_CFC_ (* Continuous Function Chart, elements in execution order *)
#0 OR(SHU6_PV1_YA4_UP_RESET, SHU6_PV1_SB)
#1 SEL(SHU6_PV1_YA4_AI1_FILTER_ON, T#0ms, T#2s)
#2 fb_YA3:ISTOK_ANALOGVH(enable: TRUE, rawValue: SHU6_PV1_1YA4_AI5, reset: #0, enableLimitCtrl: TRUE, ctrlVoltage: NOT SHU6_PV1_YA4_AI1_CVOLT, changeValueWithoutPower: TRUE, highRange: YA_HIGHRANGE, lowRange: YA_LOWRANGE, highLimit: SHU6_PV1_YA_HIGHLIMIT, lowLimit: SHU6_PV1_YA_LOWLIMIT, filterTime: #1, offset: ofset, delayEnable: YA_DELAY)
#3 SHU6_PV1_YA4_UP_VN <= #2.presentValue
#4 SHU6_PV1_YA4_UP_DOST <= #2.reliability
#5 Lt_otkr_zakr:ISTOK_LT(dost: #2.reliability, x: #2.presentValue, ust: 5, shkal: -, gist: 3)
#6 SHU6_PV1_YA4_ZKR <= #5.Xm
#7 gt_otkr_otr:ISTOK_GT(dost: #2.reliability, x: #2.presentValue, ust: 95, shkal: -, gist: 3)
#8 SHU6_PV1_YA4_OTK <= #7.Xb
#9 SUB(YA4_UST_VKL_STER_REG, YA4_UST_OTKL_STER_REG)
#10 fb_YA3bUST_VKL_STER_REG:ISTOK_GT(dost: #2.reliability, x: #2.presentValue, ust: YA4_UST_VKL_STER_REG, shkal: -, gist: #9)
#11 SHU6_PV1_YA4_B_UST_VKL_STER_REG <= #10.Xb
#12 SHU6_PV1_YA4_M_UST_VKL_STER_REG <= #10.XbN
#13 SUB(YA4_UST_OTKL_UVEL_CHAST, YA4_UST_VKL_UVEL_CHAST)
#14 fb_YA3mOTKL_STER_REG:ISTOK_LT(dost: #2.reliability, x: #2.presentValue, ust: YA4_UST_VKL_UVEL_CHAST, shkal: -, gist: #13)
#15 SHU6_PV1_YA4_M_UST_VKL_UVEL_CHAST <= #14.Xm
#16 SHU6_PV1_YA4_B_UST_VKL_UVEL_CHAST <= #14.XmN
_END_CFC_
(* the same logic as Structured Text *)
fb_YA3(enable := TRUE, rawValue := SHU6_PV1_1YA4_AI5, reset := SHU6_PV1_YA4_UP_RESET OR SHU6_PV1_SB, enableLimitCtrl := TRUE, ctrlVoltage := NOT SHU6_PV1_YA4_AI1_CVOLT, changeValueWithoutPower := TRUE, highRange := YA_HIGHRANGE, lowRange := YA_LOWRANGE, highLimit := SHU6_PV1_YA_HIGHLIMIT, lowLimit := SHU6_PV1_YA_LOWLIMIT, filterTime := SEL(SHU6_PV1_YA4_AI1_FILTER_ON, T#0ms, T#2s), offset := ofset, delayEnable := YA_DELAY);
SHU6_PV1_YA4_UP_VN := fb_YA3.presentValue;
SHU6_PV1_YA4_UP_DOST := fb_YA3.reliability;
Lt_otkr_zakr(dost := fb_YA3.reliability, x := fb_YA3.presentValue, ust := 5, gist := 3);
SHU6_PV1_YA4_ZKR := Lt_otkr_zakr.Xm;
gt_otkr_otr(dost := fb_YA3.reliability, x := fb_YA3.presentValue, ust := 95, gist := 3);
SHU6_PV1_YA4_OTK := gt_otkr_otr.Xb;
fb_YA3bUST_VKL_STER_REG(dost := fb_YA3.reliability, x := fb_YA3.presentValue, ust := YA4_UST_VKL_STER_REG, gist := YA4_UST_VKL_STER_REG - YA4_UST_OTKL_STER_REG);
SHU6_PV1_YA4_B_UST_VKL_STER_REG := fb_YA3bUST_VKL_STER_REG.Xb;
SHU6_PV1_YA4_M_UST_VKL_STER_REG := fb_YA3bUST_VKL_STER_REG.XbN;
fb_YA3mOTKL_STER_REG(dost := fb_YA3.reliability, x := fb_YA3.presentValue, ust := YA4_UST_VKL_UVEL_CHAST, gist := YA4_UST_OTKL_UVEL_CHAST - YA4_UST_VKL_UVEL_CHAST);
SHU6_PV1_YA4_M_UST_VKL_UVEL_CHAST := fb_YA3mOTKL_STER_REG.Xm;
SHU6_PV1_YA4_B_UST_VKL_UVEL_CHAST := fb_YA3mOTKL_STER_REG.XmN;
END_PROGRAM

(* POU Input/CI/MP1_OB, CFC *)
PROGRAM MP1_OB
VAR
	fb_M1_OBRbSM: ISTOK_GT;
	fb_M1b30: ISTOK_GT;
	fb_M1_OBRb45: ISTOK_GT;
	fb_M1_OBRm0_1: ISTOK_LT;
	fb_M_OBR: ISTOK_ANALOGVH;
	ofset: INT := 0;
	SR_DOST_M1: RS;
	dost_ton: TON;
END_VAR
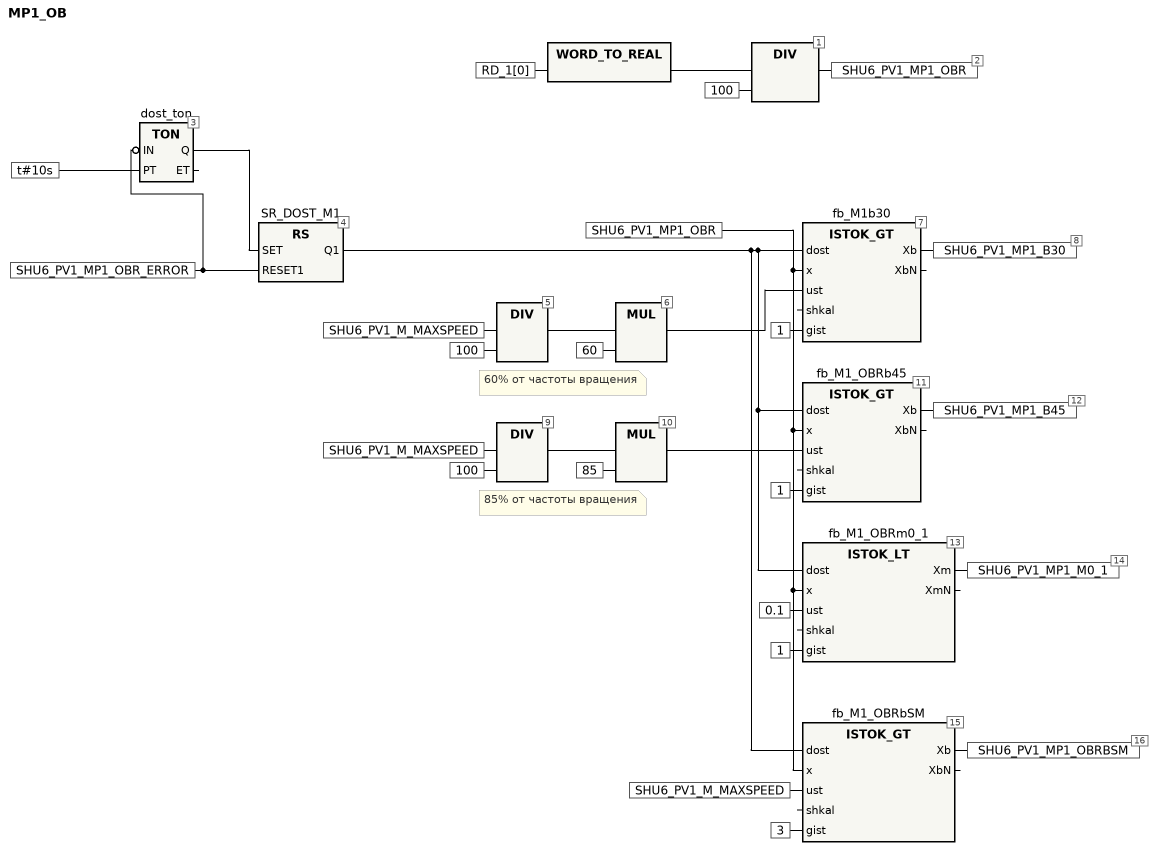
_CFC_ (* Continuous Function Chart, elements in execution order *)
(* 85% от частоты вращения *)
(* 60% от частоты вращения *)
#0 WORD_TO_REAL(RD_1[0])
#1 DIV(#0, 100)
#2 SHU6_PV1_MP1_OBR <= #1
#3 dost_ton:TON(IN: NOT SHU6_PV1_MP1_OBR_ERROR, PT: t#10s)
#4 SR_DOST_M1:RS(SET: #3.Q, RESET1: SHU6_PV1_MP1_OBR_ERROR)
#5 DIV(SHU6_PV1_M_MAXSPEED, 100)
#6 MUL(#5, 60)
#7 fb_M1b30:ISTOK_GT(dost: #4.Q1, x: SHU6_PV1_MP1_OBR, ust: #6, shkal: -, gist: 1)
#8 SHU6_PV1_MP1_B30 <= #7.Xb
#9 DIV(SHU6_PV1_M_MAXSPEED, 100)
#10 MUL(#9, 85)
#11 fb_M1_OBRb45:ISTOK_GT(dost: #4.Q1, x: SHU6_PV1_MP1_OBR, ust: #10, shkal: -, gist: 1)
#12 SHU6_PV1_MP1_B45 <= #11.Xb
#13 fb_M1_OBRm0_1:ISTOK_LT(dost: #4.Q1, x: SHU6_PV1_MP1_OBR, ust: 0.1, shkal: -, gist: 1)
#14 SHU6_PV1_MP1_M0_1 <= #13.Xm
#15 fb_M1_OBRbSM:ISTOK_GT(dost: #4.Q1, x: SHU6_PV1_MP1_OBR, ust: SHU6_PV1_M_MAXSPEED, shkal: -, gist: 3)
#16 SHU6_PV1_MP1_OBRBSM <= #15.Xb
_END_CFC_
(* the same logic as Structured Text *)
(* 85% от частоты вращения *)
(* 60% от частоты вращения *)
SHU6_PV1_MP1_OBR := WORD_TO_REAL(RD_1[0]) / 100;
dost_ton(IN := NOT SHU6_PV1_MP1_OBR_ERROR, PT := t#10s);
SR_DOST_M1(SET := dost_ton.Q, RESET1 := SHU6_PV1_MP1_OBR_ERROR);
fb_M1b30(dost := SR_DOST_M1.Q1, x := SHU6_PV1_MP1_OBR, ust := (SHU6_PV1_M_MAXSPEED / 100) * 60, gist := 1);
SHU6_PV1_MP1_B30 := fb_M1b30.Xb;
fb_M1_OBRb45(dost := SR_DOST_M1.Q1, x := SHU6_PV1_MP1_OBR, ust := (SHU6_PV1_M_MAXSPEED / 100) * 85, gist := 1);
SHU6_PV1_MP1_B45 := fb_M1_OBRb45.Xb;
fb_M1_OBRm0_1(dost := SR_DOST_M1.Q1, x := SHU6_PV1_MP1_OBR, ust := 0.1, gist := 1);
SHU6_PV1_MP1_M0_1 := fb_M1_OBRm0_1.Xm;
fb_M1_OBRbSM(dost := SR_DOST_M1.Q1, x := SHU6_PV1_MP1_OBR, ust := SHU6_PV1_M_MAXSPEED, gist := 3);
SHU6_PV1_MP1_OBRBSM := fb_M1_OBRbSM.Xb;
END_PROGRAM

(* POU Input/CI/MV1_OB, CFC *)
PROGRAM MV1_OB
VAR
	ofset: INT := 0;
	dost_ton_3: TON;
	SR_DOST_MV1: RS;
	fb_MV1b30: ISTOK_GT;
	fb_MV1_OBRb45: ISTOK_GT;
	fb_MV1_OBRm0_1: ISTOK_LT;
	fb_MV1_OBRbSM: ISTOK_GT;
END_VAR
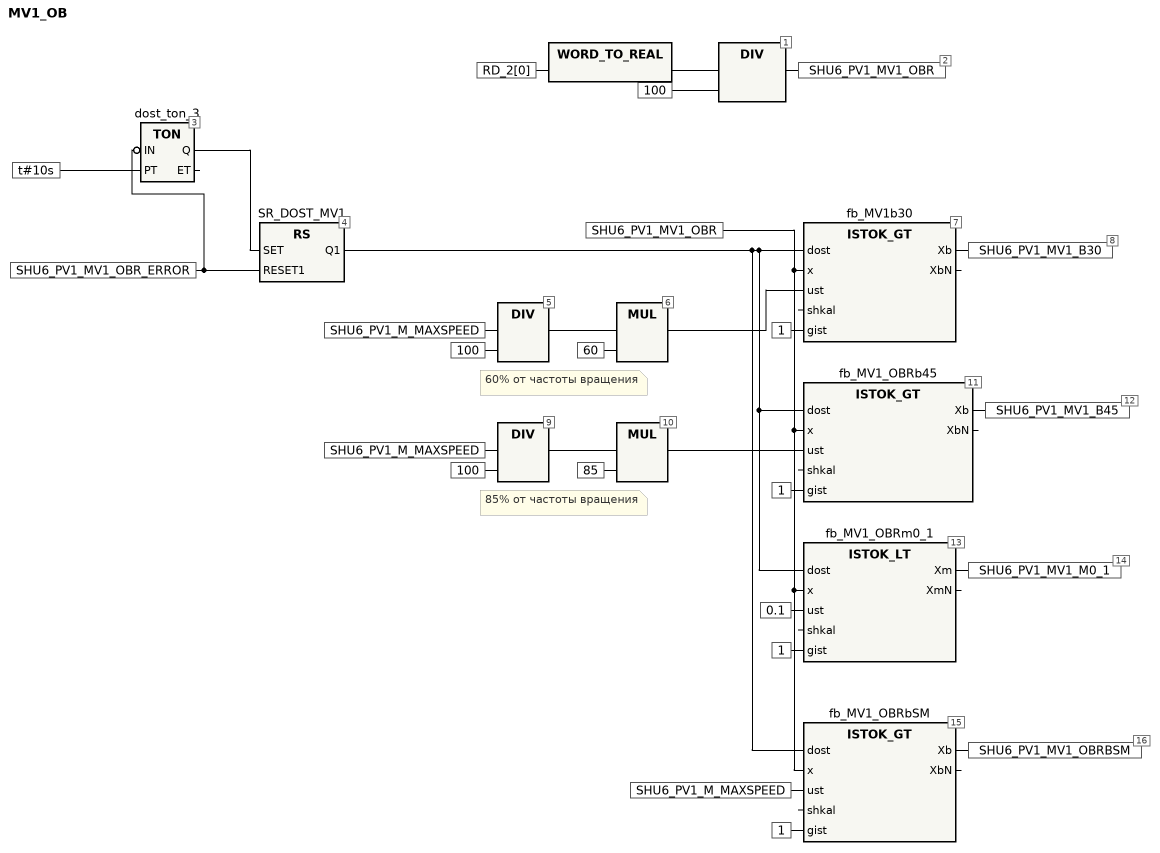
